// FB_RecipeHeaderHandler: Extracts metadata from a recipe JSON file and fills one entry in GVL_Recipe.aAvailableFiles
FUNCTION_BLOCK FB_RecipeHeaderHandler
VAR_INPUT
	sFileName       : STRING(255);
    iTargetIndex    : INT; // Index to write into array GVL_Recipe.aAvailableFiles
    bExecute        : BOOL;
END_VAR
VAR_OUTPUT
	bBusy  : BOOL;
    bError : BOOL;
    bDone  : BOOL;
    nErrId : UDINT;
END_VAR
VAR
	iStep         : INT;
    hFile         : UINT;
    sBuffer       : STRING(4096);
    fbFileOpen    : FB_FileOpen;
    fbFileRead    : FB_FileRead;
    fbFileClose   : FB_FileClose;
    fbJson        : FB_JsonDomParser;
    jsonDoc       : SJsonValue;
    jsonProp      : SJsonValue;
	bExecutePrev : BOOL; 
    bStart       : BOOL;
END_VAR

bStart := bExecute AND NOT bExecutePrev;
bExecutePrev := bExecute;

CASE iStep OF

0:
     IF bExecute THEN //bStart
        //bBusy := TRUE;
        bDone := FALSE;
        bError := FALSE;
        nErrId := 0;

        fbFileOpen(
            sNetId := '',
            sPathName := sFileName,
            nMode := FOPEN_MODEREAD OR FOPEN_MODETEXT,
            bExecute := TRUE,
			hFile => hFile
        );
		IF NOT fbFileOpen.bBusy AND NOT fbFileOpen.bError THEN
			iStep := 10;
		END_IF
        
    END_IF

10:
    fbFileOpen(
        sNetId := '',
        sPathName := sFileName,
        nMode := FOPEN_MODEREAD OR FOPEN_MODETEXT,
        bExecute := FALSE
    );
    IF NOT fbFileOpen.bBusy THEN
        IF fbFileOpen.bError THEN
            bError := TRUE;
            nErrId := fbFileOpen.nErrId;
            iStep := 100;
        ELSE
            hFile := fbFileOpen.hFile;
            fbFileRead(
                sNetId := '',
                hFile := hFile,
                pReadBuff := ADR(sBuffer),
                cbReadLen := SIZEOF(sBuffer),
                bExecute := TRUE
            );
            iStep := 20;
        END_IF
    END_IF

20:
    fbFileRead(
        sNetId := '',
        hFile := hFile,
        pReadBuff := ADR(sBuffer),
        cbReadLen := SIZEOF(sBuffer),
        bExecute := FALSE
    );
    IF NOT fbFileRead.bBusy THEN
        IF fbFileRead.bError THEN
            bError := TRUE;
            nErrId := fbFileRead.nErrId;
            iStep := 100;
        ELSE
            fbFileClose(
                sNetId := '',
                hFile := hFile,
                bExecute := TRUE
            );
            iStep := 30;
        END_IF
    END_IF

30:
    fbFileClose(
        sNetId := '',
        hFile := hFile,
        bExecute := FALSE
    );
    IF NOT fbFileClose.bBusy THEN
        IF fbFileClose.bError THEN
            bError := TRUE;
            nErrId := fbFileClose.nErrId;
            iStep := 100;
        ELSE
            jsonDoc := fbJson.ParseDocument(sBuffer);
            IF jsonDoc = 0 THEN
                bError := TRUE;
                nErrId := 16#F1000001; // Custom error code for invalid JSON
                iStep := 100;
            ELSE
                iStep := 40;
            END_IF
        END_IF
    END_IF

40:
    // Extract sCreatedBy
    jsonProp := fbJson.FindMemberPath(jsonDoc, 'stInfo/sCreatedBy');
    GVL_Recipe.aAvailableFiles[iTargetIndex].sCreatedBy := fbJson.GetString(jsonProp);

    // Extract dCreationDate
    jsonProp := fbJson.FindMemberPath(jsonDoc, 'stInfo/dCreationDate');
    GVL_Recipe.aAvailableFiles[iTargetIndex].dCreationDate := STRING_TO_DATE(fbJson.GetString(jsonProp));

    // Extract iRevision
    jsonProp := fbJson.FindMemberPath(jsonDoc, 'stInfo/iRevision');
    GVL_Recipe.aAvailableFiles[iTargetIndex].iRevision := TO_INT(fbJson.GetInt(jsonProp));

    iStep := 100;

100:
    bBusy := FALSE;
    bDone := TRUE;
    IF NOT bExecute THEN
        iStep := 0;
    END_IF

END_CASE

END_FUNCTION_BLOCK

(* stored: Version 1.1.0.1, ProductVersion 3.1.4024.12
   POU FB_RecipeHeaderHandler: Id {3a282dd4-91de-4b2b-b71c-941e4b67bb20}, SpecialFunc None *)
